FUNCTION_BLOCK TEMP_CTRL_ON_OFF_EXT
VAR_INPUT
	REAL_SV			: REAL;
	REAL_HYS			: REAL;
	REAL_HAL			: REAL;
	REAL_T_READY		: REAL; (*Value set base on -X*)
	TOutOfRangeNegative	: REAL; (*Value set base on +/- X*)
	TOutOfRangePositive	: REAL;
	INT_PV				: INT;

END_VAR


VAR_OUTPUT
	REAL_PV : REAL;
	OUT_BOOL: BOOL;
	HAL_BOOL: BOOL;
	T_READY_BOOL: BOOL;
	T_OutOfRange_BOOL : BOOL;
END_VAR

VAR

	TREADY_TEMP: REAL;
	HYS_TEMP: REAL;
	ALWAYS_OFF: BOOL;
	ALWAYS_ON_BOOL: BOOL;
	T1: TON;
	PLS1: R_TRIG;
	RS1: RS;

END_VAR

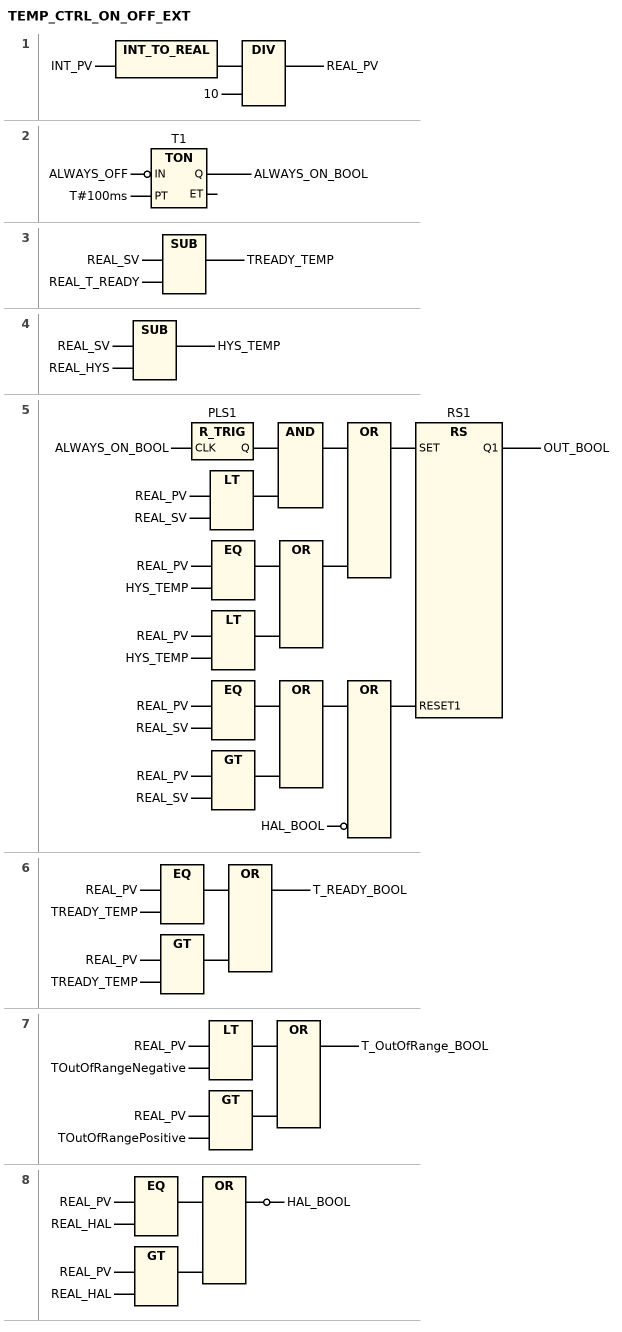
// NETWORK 1
REAL_PV := INT_TO_REAL(INT_PV) / 10;

// NETWORK 2
T1(IN := NOT ALWAYS_OFF, PT := T#100ms); // TON
ALWAYS_ON_BOOL := T1.Q;

// NETWORK 3
TREADY_TEMP := REAL_SV - REAL_T_READY;

// NETWORK 4
HYS_TEMP := REAL_SV - REAL_HYS;

// NETWORK 5
PLS1(CLK := ALWAYS_ON_BOOL); // R_TRIG
RS1(SET := PLS1.Q AND REAL_PV < REAL_SV OR (REAL_PV = HYS_TEMP OR REAL_PV < HYS_TEMP), RESET1 := (REAL_PV = REAL_SV OR REAL_PV > REAL_SV) OR NOT HAL_BOOL); // RS
OUT_BOOL := RS1.Q1;

// NETWORK 6
T_READY_BOOL := REAL_PV = TREADY_TEMP OR REAL_PV > TREADY_TEMP;

// NETWORK 7
T_OutOfRange_BOOL := REAL_PV < TOutOfRangeNegative OR REAL_PV > TOutOfRangePositive;

// NETWORK 8
HAL_BOOL := NOT (REAL_PV = REAL_HAL OR REAL_PV > REAL_HAL);

END_FUNCTION_BLOCK

(* stored: Version 1.1.0.1, ProductVersion 3.1.4024.12
   POU TEMP_CTRL_ON_OFF_EXT: Id {a9c46e37-f030-449f-a7f8-1bb3ba1625ed}, SpecialFunc None *)
